PROGRAM X10_xFastOutputs
VAR
	fbCamera01Out				: FB_IO2_OutputCtrl;
	fbCamera06Out				: FB_IO2_OutputCtrl;
END_VAR

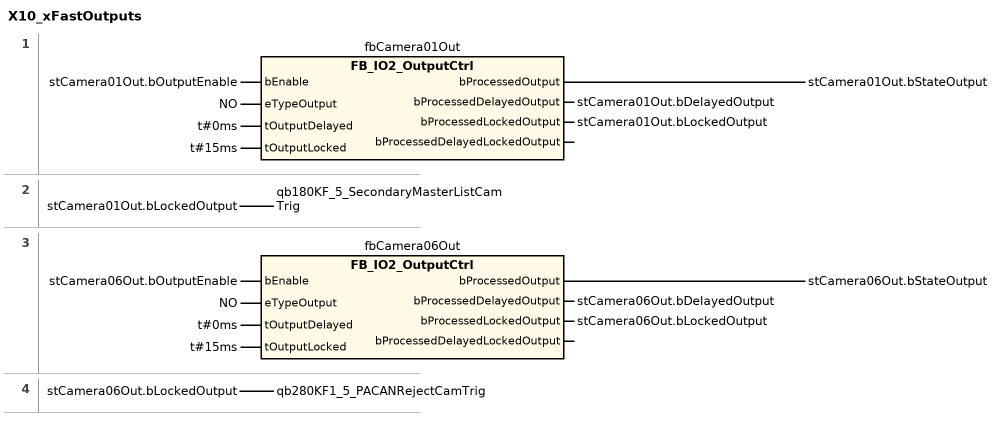
// NETWORK 1
fbCamera01Out(
    bEnable := stCamera01Out.bOutputEnable,
    eTypeOutput := NO,
    tOutputDelayed := t#0ms,
    tOutputLocked := t#15ms,
    bProcessedDelayedOutput => stCamera01Out.bDelayedOutput,
    bProcessedLockedOutput => stCamera01Out.bLockedOutput); // FB_IO2_OutputCtrl
stCamera01Out.bStateOutput := fbCamera01Out.bProcessedOutput;

// NETWORK 2
qb180KF_5_SecondaryMasterListCamTrig := stCamera01Out.bLockedOutput;

// NETWORK 3
fbCamera06Out(
    bEnable := stCamera06Out.bOutputEnable,
    eTypeOutput := NO,
    tOutputDelayed := t#0ms,
    tOutputLocked := t#15ms,
    bProcessedDelayedOutput => stCamera06Out.bDelayedOutput,
    bProcessedLockedOutput => stCamera06Out.bLockedOutput); // FB_IO2_OutputCtrl
stCamera06Out.bStateOutput := fbCamera06Out.bProcessedOutput;

// NETWORK 4
qb280KF1_5_PACANRejectCamTrig := stCamera06Out.bLockedOutput;

END_PROGRAM

(* stored: Version 1.1.0.1, ProductVersion 3.1.4024.15
   POU X10_xFastOutputs: Id {a0cd4f59-07e4-4c8a-9b61-c8734977cb18}, SpecialFunc None *)
